// SIMATIC S7-200 project (STEP 7-Micro/WIN), CPU 221 REL 01.10

SYMBOL_TABLE USER1
Start            I0.0
estop            I0.1
DC               Q0.0
Re               I0.2
END_SYMBOL_TABLE

ORGANIZATION_BLOCK MAIN:OB1
TITLE=PROGRAM COMMENTS
BEGIN
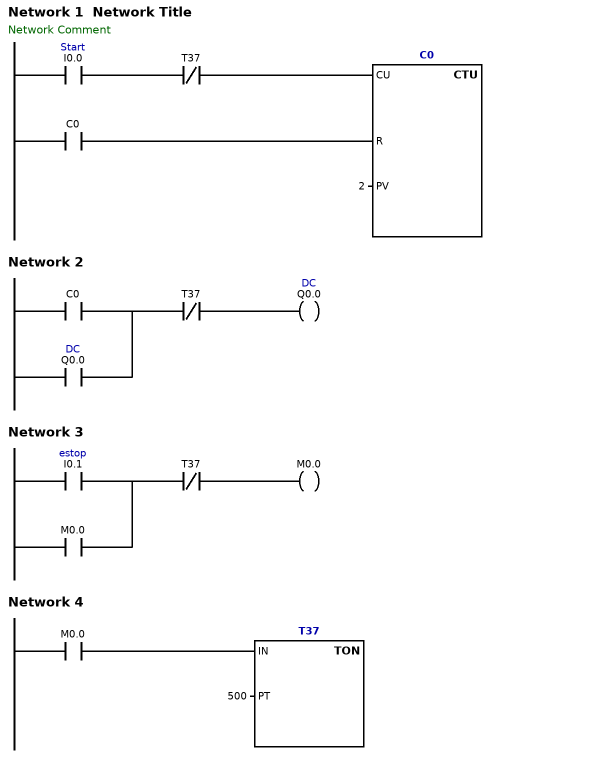
Network 1 // Network Title
// Network Comment
LD     Start:I0.0
AN     T37
LD     C0
CTU    C0, 2
Network 2
LD     C0
O      DC:Q0.0
AN     T37
=      DC:Q0.0
Network 3
LD     estop:I0.1
O      M0.0
AN     T37
=      M0.0
Network 4
LD     M0.0
TON    T37, 500
END_ORGANIZATION_BLOCK
